// TIA Portal V20 export
DATA_BLOCK "Hmi"   // DB4
// stored: MemoryReserve 100
   VAR
      mainHeader : Array[0.."NO_OF_PANELS"] of "LAF_typeHeader";   // Input from the status bar of the HMI
      operationInterlock : "LAF_typeOperationInterlockInterface";
      TestBit { S7_SetPoint := 'True'} : Array[0..9] of Bool;
   END_VAR
BEGIN
   mainHeader[0..1].hmiToPlc.acknowledge := FALSE;
   mainHeader[0..1].hmiToPlc.powerCommands := 16#00;
   mainHeader[0..1].hmiToPlc.selectedUnits := 16#0001;
   mainHeader[0..1].hmiToPlc.modeRequests := 16#0000;
   mainHeader[0..1].hmiToPlc.stateCommands := 16#0000;
   mainHeader[0..1].hmiToPlc.specialFunctions := 16#0000;
   mainHeader[0..1].plcToHmi.powerStatus := 0;
   mainHeader[0..1].plcToHmi.displayedMode := 2;
   mainHeader[0..1].plcToHmi.displayedState := 2;
   mainHeader[0..1].plcToHmi.modeRequestsButtons.visibility := 16#000F;
   mainHeader[0].plcToHmi.modeRequestsButtons.operatorControlAllowed := 16#000F;
   mainHeader[1].plcToHmi.modeRequestsButtons.operatorControlAllowed := 16#0001;
   mainHeader[0..1].plcToHmi.modeRequestsButtons.active := 16#0002;
   mainHeader[0].plcToHmi.stateCommandsButtons.visibility := 16#0000;
   mainHeader[1].plcToHmi.stateCommandsButtons.visibility := 16#000F;
   mainHeader[0..1].plcToHmi.stateCommandsButtons.operatorControlAllowed := 16#0084;
   mainHeader[0..1].plcToHmi.stateCommandsButtons.active := 16#0000;
   mainHeader[0].plcToHmi.specialFunctionButtons.visibility := 16#701fffff;
   mainHeader[1].plcToHmi.specialFunctionButtons.visibility := 16#0007;
   mainHeader[0].plcToHmi.specialFunctionButtons.operatorControlAllowed := 16#701fffff;
   mainHeader[1].plcToHmi.specialFunctionButtons.operatorControlAllowed := 16#000F;
   mainHeader[0..1].plcToHmi.specialFunctionButtons.active := 16#0000;
   operationInterlock.commands.reqMaintenanceLock := FALSE;
   operationInterlock.commands.reqMaintenanceReset := FALSE;
   operationInterlock.commands.serverMachineName := WSTRING#'ucp-3013893F1460';
   operationInterlock.commands.localMachineName := WSTRING#'Controlroom Client';
   operationInterlock.monitoring.maintenanceLockActive := FALSE;
END_DATA_BLOCK
